TYPE ST_HMIitfStructCommandTester :
STRUCT
	bInitial			:BOOL;
	bInitialTest		:BOOL;
	bProcess			:BOOL;
	bProcessHaltMode	:BOOL;
	bProcessHaltStep	:BOOL;
	bCmdFeedback		:BOOL;
	
	
	
	
END_STRUCT
END_TYPE

(* stored: Version 1.1.0.1, ProductVersion 3.1.4024.16
   DUT ST_HMIitfStructCommandTester: Id {0507080a-756d-4d1d-bd8f-a0b0866f7553} *)
